FUNCTION FC_GetMaxLapTime : TIME
VAR_IN_OUT
	// Last 10 lap times
	aLapTimes: ARRAY[0..10] OF TIME;
END_VAR
VAR
	nIndex: INT;
END_VAR

aLapTimes[0] := T#0S;

FOR nIndex := 1 TO 10 DO
    // Compare current max value with index
    IF aLapTimes[nIndex] > aLapTimes[0] THEN
        // Store new max value
        aLapTimes[0] := aLapTimes[nIndex];
    END_IF
END_FOR

FC_GetMaxLapTime := aLapTimes[0];

END_FUNCTION

(* stored: Version 1.1.0.1
   POU FC_GetMaxLapTime: Id {4e32b790-012b-4c2d-88b1-1c27f1a55e47}, SpecialFunc None *)
